{attribute 'qualified_only'}
{attribute 'strict'}
TYPE E_ScannerStatus :
(
	Offline := 0,
	Online := 1,
	Ready := 2,
	Busy := 3,
	Faulted := 4
);
END_TYPE

(* stored: Version 1.1.0.1, ProductVersion 3.1.4022.10
   DUT E_ScannerStatus: Id {30ed4dbe-2531-467e-837c-e3939188581f} *)
